Fanuc TP program (LS listing): _ZERO.LS

/PROG  _ZERO
/ATTR
OWNER		= MNEDITOR;
COMMENT		= "";
PROG_SIZE	= 228;
CREATE		= DATE 23-08-30  TIME 16:45:20;
MODIFIED	= DATE 23-09-08  TIME 08:34:50;
FILE_NAME	= ;
VERSION		= 0;
LINE_COUNT	= 2;
MEMORY_SIZE	= 600;
PROTECT		= READ_WRITE;
TCD:  STACK_SIZE	= 0,
      TASK_PRIORITY	= 50,
      TIME_SLICE	= 0,
      BUSY_LAMP_OFF	= 0,
      ABORT_REQUEST	= 0,
      PAUSE_REQUEST	= 0;
DEFAULT_GROUP	= 1,*,*,*,*;
CONTROL_CODE	= 00000000 00000000;
LOCAL_REGISTERS	= 0,0,0;
/APPL
/APPL

AUTO_SINGULARITY_HEADER;
  ENABLE_SINGULARITY_AVOIDANCE   : TRUE;

PLTZ_MODE_HEADER;
 PLTZ_MODE_ENABLE   : FALSE;
 J4TURN  : ZERORAD;
 ORIENT  : DOWNWARDS;
/MN
   1:  CALL _MOVE_TO_UF(1) ;
   2:   ;
/POS
/END
